(* CODESYS project lclsgeneral.library
   Author: Alex Wallace
   Placeholder: LCLS General
   Title: LCLS General
   Version: 0.0.0
   Description: Generally useful POUs:
      - Logger
      - FB diagnostics
      - EtherCAT diagnostic
   Company: SLAC

Project tree, tasks and I/O mapping:
  libraries: Tc2_EtherCAT, * (Beckhoff Automation GmbH); Tc2_ModbusSrv, * (Beckhoff Automation GmbH); Tc2_Standard, * (Beckhoff Automation GmbH); Tc2_System, * (Beckhoff Automation GmbH); Tc2_TcpIp, * (Beckhoff Automation GmbH); Tc2_Utilities, * (Beckhoff Automation GmbH)
  Data types/
    Misc/
      data type ST_EcDevice
      data type ST_FbDiagnostics
      data type ST_System
  Diagnostics/
  GVLs/
    global variables DefaultGlobals
  POUs/
    Functions/
      function block FB_EcatDiag [ST]
      function block FB_Index [ST]: Dec, DecVal, Inc, IncVal
      function block FB_XKoyoPLCModbus [ST]
    Logger/
      DUTs/
        data type E_MesgSevr
        data type E_MessengerState
        data type E_Subsystem
      function block FB_Logger [ST]: Manager, SocketSendTo
      function block FB_LogMessage [ST]
      global variables GVL_Logger
      function SYSTEM_TIME_TO_RFC3339 [ST]
*)

// Data types/Misc/ST_EcDevice
//EtherCAT Device struct for EtherCAT diagnostics
TYPE ST_EcDevice :
STRUCT
	nDeviceState: BYTE; //EtherCAT state machine state number, 8 is OP is good
	sDeviceState :STRING; //EtherCAT state machine state, OP is good
	nLinkState: BYTE; //EtherCAT link state, 8 is good
	nAddrr: WORD; //EtherCAT slave address
	sType: STRING; //EtherCAT slave type
	sName:STRING; //EtherCAT slave name
END_STRUCT
END_TYPE

// Data types/Misc/ST_FbDiagnostics
//Stuff to log messages within function blocks
TYPE ST_FbDiagnostics :
STRUCT
	asResults	:	ARRAY [1..20] OF T_MaxString; //Diagnostic messages, use to record state changes or other important events.
	{attribute 'naming' := 'omit'}
	//Incrementer, included here to facilitate using asResults
	resultIdx	:	FB_Index := ( 
		LowerLimit := 1,
		UpperLimit := 20
	);
	{attribute 'naming' := 'omit'}
	fString	:	FB_FormatString; //Use to create good log messages, similar to C++ fstring
END_STRUCT
END_TYPE

// Data types/Misc/ST_System
//Defacto system structure, must be included in all projects
TYPE ST_System :
STRUCT
	
	xSwAlmRst 		: BOOL;(* Global Alarm Reset - EPICS Command *)
	xAtVacuum 	    : BOOL;(* System At Vacuum *)
	xFirstScan	    : BOOL; (* This boolean is true for the first scan, and is false thereafter, use for initialization of stuff *)
	xOverrideMode	: BOOL; //This bit is set when using the override features of the system
	xIOState        : BOOL; (* ECat Bus Health *)
	{attribute 'naming' := 'omit'}
	I_EcatMaster1 AT %I* : AMSNETID; (* AMS Net ID used for FB_EcatDiag, among others *)

END_STRUCT
END_TYPE

// POUs/Logger/DUTs/E_MesgSevr
//Syslog message severities
{attribute 'flags'}
TYPE E_MesgSevr :
(
	Emergency := 0, //system is unusable
	Alert	:= 1,	//action must be taken immediately
	Critical:= 2,	//critical conditions
	Error	:= 3,	//error conditions
	Warning	:= 4,	//warning conditions
	Notice	:= 5,	//normal but significant condition
	Info	:= 6,	//informational messages
	Debug	:= 7	//debug-level messages
) WORD;
END_TYPE

// POUs/Logger/DUTs/E_MessengerState
//State of the FB_Logger
TYPE E_MessengerState :
(
	Init := 0, //Messenger is not yet initialized
	CreateSocket	:= 1, //Messenger is opening the connection to the syslog server
	Active	:= 2, //Messenger is running, shipping messages to syslog
	CloseSocket := 3, //Messenger is closing the connection to the syslog server
	Err	:= 10 //Messenger has hit some error. Check diagnostics structure in the FB, this always goes back to Init.
);
END_TYPE

// POUs/Logger/DUTs/E_Subsystem
//LCLS Defined subsystems, make sure these correspond with casSubsystems in FB_LogMessage
TYPE E_Subsystem :
(
	NILVALUE := 0, //Undefined system
	VACUUM := 1, //Vacuum control system
	MPS := 2, //Machine protection system
	MOTION := 3, //Motion control systems
	FIELDBUS := 4, //EtherCAT networks
	SDS := 5 //Sample delivery system
)WORD;
END_TYPE

// GVLs/DefaultGlobals
//These are variables every PLC project should have
VAR_GLOBAL
	
	stSys	:	ST_System; //Included for you
END_VAR

// POUs/Logger/GVL_Logger
{attribute 'qualified only'}
//Global variables for logging to syslog
VAR_GLOBAL CONSTANT
	csNILVALUE	:	STRING(1) := '-'; //Syslog standard placeholder/ blank
	{attribute 'analysis' := '-33'} //This is used just below in decl. of asLoggerMesgBuffer
	cnLoggerMesgArraySize : INT := 50; //Size of the Logger buffer
	// Syslog Version
	cnSyslogVer: WORD := 1; //Logger written to work with Syslog V1
END_VAR
VAR_GLOBAL
	asLoggerMesgBuffer	:	ARRAY [0..cnLoggerMesgArraySize] OF T_MaxString; //Logger message buffer, FB_LogMessage puts messages in here for FB_Logger to send out
	gsCurrentTime	:	T_MaxString := csNILVALUE; //For timestamping messages
	{analysis -33}
	fbLogMessage : FB_LogMessage; //Instantiated here to be used everywhere
	{analysis +33}
	fbLoggerBuffer 			:	FB_StringRingBuffer; //For working with the Logger message buffer
	
	//Note: FB_Logger is not declared here as it needs to be integrated into each project manually. See FB comment for more info.
END_VAR

// POUs/Functions/FB_EcatDiag
(* 
Ecat bus diagnostic tool
2015-11-4 Alex Wallace
This function block checks the states of all slaves on the ecat bus network, 
it could be modified to export the states of the slaves on an individual basis,
but for now it sets the output boolean true if all slaves are OP and false otherwise.
To start the block provide a falling edge on the first pass boolean input.

2018-05-05 Margaret Ghaly
Function block has been modified to retrieve the Device State of the Ethercat Master.
It also exports the states and information of each individual configured Slave. 
And saves them in the array q_aEcConfSlaveInfo.
*)
FUNCTION_BLOCK FB_EcatDiag
VAR_INPUT
	{attribute 'naming' := 'omit'}
	I_AMSNetId AT %I* : AMSNETID; //Link to the AMSNETID name in the ethercat master info.
	i_xFirstPass: BOOL; //Hook to system first pass boolean for proper intialization (must be true for the first cycle of the PLC)
END_VAR
VAR_OUTPUT
	q_xAllSlaveStatesGood: BOOL; // Set to True if all Slaves are in OP State
	q_anTermStates: ARRAY[1..256] OF BYTE; //ECAT State of terminals in the bus
	q_xMasterStateGood:BOOL; // Set to True if the Master Device State is OP
	q_nMasterState: WORD; // The Device State of the Master
	q_sMasterState:STRING; //State of the ECAT master
	q_astEcConfSlaveInfo :  ARRAY[1..256] OF ST_EcDevice; //State of all ECAT slaves in the bus
	q_nSlaves: UINT; // the Number of the connected Slaves
END_VAR
VAR
	sNetId: T_AmsNetId; //NetId string
	astTermStates: ARRAY[1..256] OF ST_EcSlaveState; //ECAT Slave States Buffer
	astEcConfSlaveInfo: ARRAY[1..256] OF ST_EcSlaveConfigData; //ECAT Slave Configs Buffer
	fbGetAllSlaveStates: FB_EcGetAllSlaveStates; //Acquires the ECAT Slave States puts them into astTermStates 
	
	fbGetMasterState: FB_EcGetMasterState; //Acquires ECAT Master State
	fbGetConfSlaves: FB_EcGetConfSlaves; //Acquires the ECAT slave configuration of the bus (how many, what kind, etc)
	{attribute 'naming' := 'omit'} 
	ftReset: F_TRIG; //Reset trigger sensor
	{attribute 'naming' := 'omit'}
	ftMasterReset: F_TRIG; //Retrigger sensor for GetMasterState
	nIterator: INT; //Generic iterator placeholder
END_VAR

//Create the net ID string
sNetId := F_CreateAmsNetId(I_AMSNetId);

//Query the state of all terminals, collect in astTermStates
ftReset(CLK:=fbGetAllSlaveStates.bBusy OR i_xFirstPass);
fbGetAllSlaveStates.bExecute := ftReset.Q;
fbGetAllSlaveStates(sNetId:=sNetId, pStateBuf := ADR(astTermStates), cbBufLen:=SIZEOF(astTermStates));
//Keep checking...



//Cycle through each entry in the array and check if we have anyone not in OP and that the link state is good.
// If so, then set our global IO bad boolean.
IF fbGetAllSlaveStates.nSlaves > 0 THEN
	q_xAllSlaveStatesGood := TRUE;
FOR nIterator := 1 TO (UINT_TO_INT(fbGetAllSlaveStates.nSlaves) ) BY 1
	DO
	IF NOT( (astTermStates[nIterator].deviceState = EC_DEVICE_STATE_OP) AND (astTermStates[nIterator].linkState = EC_LINK_STATE_OK)) THEN
		q_xAllSlaveStatesGood := FALSE;
	END_IF
	q_anTermStates[nIterator] := astTermStates[nIterator].deviceState;
	q_astEcConfSlaveInfo[nIterator].nDeviceState :=astTermStates[nIterator].deviceState;//
	q_astEcConfSlaveInfo[nIterator].nLinkState :=astTermStates[nIterator].linkState;//
	q_astEcConfSlaveInfo[nIterator].sDeviceState:= F_ConvSlaveStateToString(state:=astTermStates[nIterator]);//
	
END_FOR
END_IF

// Read the EtherCAT state of the master. If the call is successful, 
//the State output variable of type WORD contains the requested status information.
ftMasterReset(CLK:=fbGetMasterState.bBusy OR i_xFirstPass);
fbGetMasterState(sNetId:= sNetId, bExecute:=ftMasterReset.Q, 
				state => q_nMasterState,bError=>,
				nErrId=>);
q_xMasterStateGood:= (fbGetMasterState.state = BYTE_TO_UINT(EC_DEVICE_STATE_OP));
q_sMasterState := F_ConvMasterDevStateToString(fbGetMasterState.state);

//This function is used to read a list of all configured slaves from the EtherCat master object Directory
//needs to run only once
fbGetConfSlaves(bExecute := i_xFirstPass, sNetId :=sNetId, pArrEcConfSlaveInfo := ADR(astEcConfSlaveInfo),cbBufLen := SIZEOF(astEcConfSlaveInfo));
q_nSlaves:=fbGetConfSlaves.nSlaves;

IF  NOT (fbGetConfSlaves.bBusy) THEN
	FOR nIterator := 1 TO (UINT_TO_INT(fbGetConfSlaves.nSlaves) ) BY 1
	DO
	q_astEcConfSlaveInfo[nIterator].nAddrr :=astEcConfSlaveInfo[nIterator].nAddr;
	q_astEcConfSlaveInfo[nIterator].sName :=astEcConfSlaveInfo[nIterator].sName;
	q_astEcConfSlaveInfo[nIterator].sType :=astEcConfSlaveInfo[nIterator].sType;
END_FOR
	fbGetConfSlaves.bExecute := FALSE;
END_IF

END_FUNCTION_BLOCK

// POUs/Functions/FB_Index
(* Index FB
A. Wallace 2016-9-3

Why doesn't beckhoff have this as a builtin type?

Use this thing to have a simple indexer with rollover.

*)
FUNCTION_BLOCK FB_Index
VAR_INPUT
	{attribute 'naming' := 'off'}
	LowerLimit : INT := 1; //Incrementer will rollver over to this value (and initialize to this value)
	ValInc : INT := 1; //Incrementer increments by this value
	UpperLimit	:	INT := 1; //Incrementer will rollover at this value to lower limit
	{attribute 'naming' := 'off'}
END_VAR
VAR_OUTPUT
	
END_VAR
VAR
	nVal	:	INT := LowerLimit; //Internal incrementer value, initialized to LowerLimit
END_VAR

{analysis -2} //Only the methods and actions are needed

ACTION Dec:
nVal := nVal - ValInc;
IF nVal < LowerLimit THEN nVal := UpperLimit; END_IF
END_ACTION

//Decrement the counter and return new value
METHOD DecVal : INT
VAR_INPUT
END_VAR
Dec();
DecVal := nVal;
END_METHOD

ACTION Inc:
// Dont use this, use ValInc
nVal := nVal + ValInc;
IF nVal >  UpperLimit THEN nVal := LowerLimit; END_IF
END_ACTION

//Increment the counter and return new value
METHOD PUBLIC IncVal : INT
VAR_INPUT
END_VAR
Inc();
IncVal := nVal;
END_METHOD

END_FUNCTION_BLOCK

// POUs/Functions/FB_XKoyoPLCModbus
//Facilitates communication between Beckhoff and Koyo PLC over the network.
FUNCTION_BLOCK FB_XKoyoPLCModbus
VAR
	fbKoyo_PLCInputCoilsRx	:	FB_MBReadCoils; //FB for reading the coils from the other PLC
	anKoyo_PLC_CnBits	:	ARRAY [0..20] OF BYTE; //Buffer for coil readbacks
	{attribute 'naming' := 'omit'}
	ftReset	: F_TRIG; //Reset edge sensor
	{attribute 'naming' := 'omit'}
	tonRetry : TON; //Retry timer
	nIndex : INT; //Index for clearing the coil array
END_VAR

VAR_INPUT
	i_tRetryTime : TIME := T#10S; //Retry time if modbus transaction fails
	i_sIPAddr	 : STRING[15]; //IP address of the Koyo PLC
END_VAR

VAR_OUTPUT
	q_xNoPLCResponse : BOOL := TRUE; //Could not reach the PLC if true
	q_anPLCResponse   : ARRAY [0..20] OF BYTE; //Buffer of coils retrieved from the other PLC
	q_xError         : BOOL := FALSE; //Transaction or other error
END_VAR

(* Look ma' no wires! *)
(* A. Wallace, 2015-7-22 
XKoyoPLCModbus

Facilitates communication between Beckhoff and Koyo PLC over the network.

Useful if you don't have time to run a wire. Fairly reliable.

*)

(* Modbus Info for Koyo
Modbus Addresses for
Koyo DL05/06/240/250/260/430/440/450 PLCs
PLC Memory Type		| Modbus start address Decimal (octal) | Function codes
Inputs (X)			  2048 (04000)							2
Special Relays (SP)	  3072 (06000)							2
Outputs (Y)			  2048 (04000)							1, 5, 15
Control Relays (C)	  3072 (06000)							1, 5, 15
Timer Contacts (T)	  6144 (014000)							1, 5, 15
Counter Contacts (CT) 6400 (014400)							1, 5, 15
Stage Status Bits (S) 6144 (012000)							1, 5, 15
*)

(* Begin code *)
// Retry after some time
tonRetry.IN := NOT fbKoyo_PLCInputCoilsRx.bBusy;
tonRetry.PT := i_tRetryTime;
tonRetry();

ftReset(CLK:=fbKoyo_PLCInputCoilsRx.bBusy);
ftReset();

fbKoyo_PLCInputCoilsRx.bExecute := ftReset.Q OR tonRetry.Q;

fbKoyo_PLCInputCoilsRx(sIPAddr:='i_sIPAddr', nTCPPort:=502, nQuantity:=32, nMBAddr:=8#6000, cbLength:=USINT_TO_UDINT(SIZEOF(anKoyo_PLC_CnBits)),  pDestAddr:=ADR(anKoyo_PLC_CnBits), tTimeout:=T#10S);

//run some error code for modbus
IF fbKoyo_PLCInputCoilsRx.bError THEN
	//if there's a modbus error, set all incoming bits to zero
	{analysis -41} //There are one-liners for resetting an array to zero but they don't comply with 61131
	FOR nIndex := 0 TO USINT_TO_INT(SIZEOF(anKoyo_PLC_CnBits))-1 DO //starts at 0
		anKoyo_PLC_CnBits[nIndex]:=0;
	END_FOR
	{analysis +41}
	q_xError := TRUE;
	
ELSIF ftReset.Q AND fbKoyo_PLCInputCoilsRx.cbRead > 0 THEN
	fbKoyo_PLCInputCoilsRx.bExecute := FALSE;
	q_xNoPLCResponse:= FALSE;
	q_xError := FALSE;

//more error code cause we didn't manage to read anything	
ELSIF fbKoyo_PLCInputCoilsRx.cbRead = 0 THEN
	q_xError := TRUE;
	q_xNoPLCResponse:= TRUE;
			
END_IF

q_anPLCResponse := anKoyo_PLC_CnBits;

END_FUNCTION_BLOCK

// POUs/Logger/FB_Logger
(* Syslog Logger
A. Wallace 2016-9-3

This is used to pass PLC notification messeges to a syslog server.

This POU constantly attempts to send out messages from the global buffer: GVL_Logger.fbLoggerBuffer.
This buffer is filled by calling fbLogMessage.

NOTE: FB_Logger must integrated into your project manually. It is recommended that you add it to its own 
task.
*)
FUNCTION_BLOCK FB_Logger
VAR_INPUT
	i_xReset		:	BOOL := FALSE; //Closes the socket and attempts to open another
END_VAR
VAR
	fbUDPSocketManager	:	FB_ConnectionlessSocket; //Creates the UDP socket handle to the syslog server
	stUDPSocket			:	T_HSOCKET; //UDP socket handle for syslog server
	fbUDPSocketSend		:	FB_SocketUdpSendTo; //FB for sending the sOutgoingMesg
	sOutgoingMesg		:	T_MaxString; //Outgoing message holder
	eState				:	E_MessengerState; //State of the messenger connection to the syslog server
	stDiag				:	ST_FbDiagnostics; //Generic FB diagnostics, check here for insight into errors/ other FB events
	{attribute 'naming' := 'omit'}
	rtReset				:	R_TRIG; //Reset sensor
	fbGetSystemTime		:	FB_LocalSystemTime := (bEnable := TRUE); //Acquires system time as message is being sent
	fbGetHostName		:	FB_GetHostName := (bExecute := TRUE, sNetID := ''); //Acquires name of the PLC
	{attribute 'naming' := 'omit'}
	ctuSentSomething	:	CTU := (PV := 100); //Diagnostic to indicate this thing is working. Increments with each successful send.
	{attribute 'naming' := 'omit'}
	rtSocketSendErr		:	R_TRIG; //Socket send error sensor
	sHostName	:	T_MaxString := csNILVALUE; //PLC hostname holder
END_VAR
VAR CONSTANT
	cPSLogHost	: T_IPv4Addr := '172.21.32.9'; //syslog host
	cnUdpSyslog	:	UDINT := 514; //syslog port
END_VAR



fbLoggerBuffer.pBuffer := ADR(asLoggerMesgBuffer); 
fbLoggerBuffer.cbBuffer:= UINT_TO_UDINT(SIZEOF(asLoggerMesgBuffer));

fbGetSystemTime(); 
IF fbGetSystemTime.bValid THEN
	gsCurrentTime := SYSTEM_TIME_TO_RFC3339(fbGetSystemTime.systemTime);
ELSE
	gsCurrentTime := csNILVALUE;
END_IF

fbGetHostName();
IF NOT (fbGetHostName.bBusy OR fbGetHostName.bError) THEN
	sHostName := fbGetHostName.sHostName;
ELSE
	sHostName := csNILVALUE;
END_IF

rtReset(CLK:=i_xReset);
IF rtReset.Q THEN
	eState := E_MessengerState.CloseSocket;
END_IF

rtSocketSendErr(CLK:=fbUDPSocketSend.bError);

CASE eState OF
	E_MessengerState.Init:
		;
	E_MessengerState.CreateSocket:
		fbUDPSocketManager.nLocalPort := cnUdpSyslog;
		fbUDPSocketManager.bEnable := TRUE;
		
		IF fbUDPSocketManager.eState = E_SocketConnectionlessState.eSOCKET_CREATED THEN
			eState := E_MessengerState.Active;
		ELSIF fbUDPSocketManager.bError THEN
			eState := E_MessengerState.Err;
			fbUDPSocketManager.bEnable := FALSE;
			stDiag.fString( sOut=>stDiag.asResults[stDiag.resultIdx.IncVal()], sFormat:='Socketmanger error in createsocket: %d', arg1:=F_UDINT(fbUDPSocketManager.nErrID));
		ELSE
			eState := E_MessengerState.Err;
			stDiag.fString( sOut=>stDiag.asResults[stDiag.resultIdx.IncVal()], sFormat:='Something else happened in createsocket -> error');
		END_IF
	E_MessengerState.Active:
		IF fbUDPSocketManager.eState = E_SocketConnectionlessState.eSOCKET_TRANSIENT  OR 
			fbUDPSocketManager.bError THEN
			eState := E_MessengerState.Err; 
			stDiag.fString( sOut=>stDiag.asResults[stDiag.resultIdx.IncVal()], sFormat:='Socketmanager error in active: %d', arg1:=F_UDINT(fbUDPSocketManager.nErrID));
		END_IF
		
		// While the socket is active, go ahead and send whatever is in the buffer
		IF rtSocketSendErr.Q THEN
			eState := E_MessengerState.Err;
			stDiag.fString( sOut=>stDiag.asResults[stDiag.resultIdx.IncVal()], sFormat:='Socket send error: %d', arg1:=F_UDINT(fbUDPSocketSend.nErrId));
		ELSIF fbLoggerBuffer.nCount > 0 AND NOT fbUDPSocketSend.bBusy THEN
			fbLoggerBuffer.A_RemoveHead(getValue=>sOutgoingMesg);
			fbUDPSocketSend.bExecute := TRUE; //reset in the action after busy goes true
			IF sOutgoingMesg <> '' THEN
				ctuSentSomething(CU:=TRUE);
			END_IF
		ELSIF fbLoggerBuffer.nCount = 0 OR fbUDPSocketSend.bBusy THEN
			stDiag.fString( sOut=>stDiag.asResults[stDiag.resultIdx.IncVal()], sFormat:='Waiting to send');
			ctuSentSomething(CU:=FALSE);
		ELSE
			eState := E_MessengerState.Err;
			stDiag.fString( sOut=>stDiag.asResults[stDiag.resultIdx.IncVal()], sFormat:='Something else happened in active -> error');
		END_IF
		
	E_MessengerState.CloseSocket:
		fbUDPSocketManager.bEnable := FALSE;
		IF fbUDPSocketManager.eState = E_SocketConnectionlessState.eSOCKET_CLOSED THEN
			eState := E_MessengerState.Init;
		ELSIF fbUDPSocketManager.bBusy AND NOT fbUDPSocketManager.bEnable THEN
			;
		ELSIF fbUDPSocketManager.bError THEN
			eState := E_MessengerState.Err;
		ELSE
			eState := E_MessengerState.Err;
		END_IF
	E_MessengerState.Err:
		eState := E_MessengerState.Init;
		stDiag.asResults[stDiag.resultIdx.IncVal()] := 'Moving back to Init state from Error';
	ELSE
		eState := E_MessengerState.Init;		
		stDiag.asResults[stDiag.resultIdx.IncVal()] := 'Uncaught state';
END_CASE



Manager();
SocketSendTo();

ACTION Manager:
fbUDPSocketManager(hSocket => stUDPSocket);
END_ACTION

ACTION SocketSendTo:
fbUDPSocketSend.hSocket := stUDPSocket;
fbUDPSocketSend.sRemoteHost := cPSLogHost;
fbUDPSocketSend.nRemotePort := cnUdpSyslog;
fbUDPSocketSend.pSrc := ADR(sOutgoingMesg);
fbUDPSocketSend.cbLen := UINT_TO_UDINT(SIZEOF(sOutgoingMesg));
fbUDPSocketSend();
fbUDPSocketSend.bExecute R= fbUDPSocketSend.bBusy;
END_ACTION

END_FUNCTION_BLOCK

// POUs/Logger/SYSTEM_TIME_TO_RFC3339
//Converts Beckhoff PLC SYSTEMTIME to RFC3339 time format as a string
{attribute 'naming' := 'omit'}
{attribute 'analysis' := '-23'}
FUNCTION SYSTEM_TIME_TO_RFC3339 : STRING(255)
VAR_INPUT
	{attribute 'naming' := 'omit'}
	tCurrentTime	:	TIMESTRUCT; //TIMESTRUCT Time to convert to RFC3339
END_VAR
VAR
END_VAR

SYSTEM_TIME_TO_RFC3339 := CONCAT(REPLACE(SYSTEMTIME_TO_STRING(tCurrentTime), 'T', 1, 11), 'Z');

END_FUNCTION

// POUs/Logger/FB_LogMessage
// LogMessage
// A Wallace, 18-4-12
// Adds a message to the global queue to be sent to the syslog server
FUNCTION_BLOCK FB_LogMessage
VAR_INPUT	
	i_sMsg	:	STRING; //Message to send
	i_eSevr	:	E_MesgSevr; //Message severity
	i_eSubsystem	:	E_Subsystem; //In-lieu of App-name in the RFC-5424
END_VAR
VAR

	fbFormatString		:	FB_FormatString; //String formatter
	sPRIVAL				: 	T_MaxString := csNILVALUE; //Priority value
	sPID				: 	T_MaxString := csNILVALUE; //Unused
	sSubsystem			: 	T_MaxString := csNILVALUE; //Type of subsystem for organizing in syslog later
	nSyslogVer			: 	WORD := cnSyslogVer; //Version of syslog
	sSD					: 	T_MaxString := csNILVALUE; //Unused
	sMsg				: 	T_MaxString := csNILVALUE; //Message to send
END_VAR
VAR CONSTANT
	{attribute 'naming' := 'off'}
	i_sPID	:	STRING := csNILVALUE;	//Not currently used
	i_sMSGID	:	STRING := csNILVALUE; //Not currently used
	i_sSD	:	STRING := csNILVALUE; //Not currently used
	{attribute 'naming' := 'on'}
	casSubsystems	:	ARRAY [0..5] OF STRING := ['-', 'VACUUM', 'MPS', 'MOTION', 'FIELDBUS', 'SDS']; //LCLS defined subsystems for global logging
	cnFacility: WORD := 20; // local4
END_VAR

fbLoggerBuffer.putValue := '';
fbLoggerBuffer.pBuffer := ADR(asLoggerMesgBuffer); //Global buffer address
fbLoggerBuffer.cbBuffer := UINT_TO_UDINT(SIZEOF(asLoggerMesgBuffer));

fbFormatString.sFormat := '<%s> %d %s %s %s %s BOM%s';

sPRIVAL := LEFT( WORD_TO_STRING(cnFacility * 8 + i_eSevr), 5);
sPID := csNILVALUE;
sSubsystem := casSubsystems[i_eSubsystem];
nSyslogVer := cnSyslogVer;
sSD := i_sSD;
sMsg := i_sMsg;
//bad language ahead, sorry
fbFormatString.arg1 := F_STRING(sPRIVAL);
fbFormatString.arg2 := F_WORD(nSyslogVer);
fbFormatString.arg3 := F_STRING(gsCurrentTime);
fbFormatString.arg4 := F_STRING(sSubsystem);
fbFormatString.arg5 := F_STRING(sPID);
fbFormatString.arg6 := F_STRING(sSD);
fbFormatString.arg7 := F_STRING(sMsg);
fbFormatString( sOut=>fbLoggerBuffer.putValue);
fbLoggerBuffer.A_AddTail();

END_FUNCTION_BLOCK
